FUNCTION_BLOCK FB_MotorCoilsCtrl
VAR_INPUT
	i_Interlocks		:ARRAY[1..8] OF BOOL;
	i_AutoCmdSlow		:BOOL;
	i_AutoCmdFast		:BOOL;
	i_ManCmdSlow		:BOOL;
	i_ManCmdFast		:BOOL;
	i_ManStop			:BOOL;
	i_SlowSpeed			:REAL;
	i_FastSpeed			:REAL;
	i_Feedback1AP		:REAL;
	i_Feedback2AP		:REAL;
	i_EnableMonitor		:BOOL;
	i_MonitorTime		:INT;
	i_MonitorTolerance	:INT;
	i_ServiceMode		:BOOL;
	i_MaintLimit		:REAL;
	i_PresetValue		:REAL;
	i_WritePreset		:BOOL;
END_VAR
VAR_OUTPUT
	q_InterlocksOK		:BOOL;
	q_bCmdSlow			:BOOL;
	q_bCmdFast			:BOOL;
	q_FeedbackMonFlt	:BOOL;
	q_TotalHours		:REAL;
	q_MaintHours		:REAL;
	q_bMaintCall		:BOOL;	
	q_State				:INT;
END_VAR
VAR
	bInTolerance		:BOOL;
	tRunTime			:TIME;
	rRunTime			:REAL;
	tonMonFdb			:TON;
	tonMotorRun			:TON;
	tofMotorRun			:TOF;
END_VAR
VAR // added by the converter: edge detectors and wires of the graphical bodies
    _w1, _w2 : BOOL;
    _ft1, _ft2 : F_TRIG;
    _rt1 : R_TRIG;
END_VAR

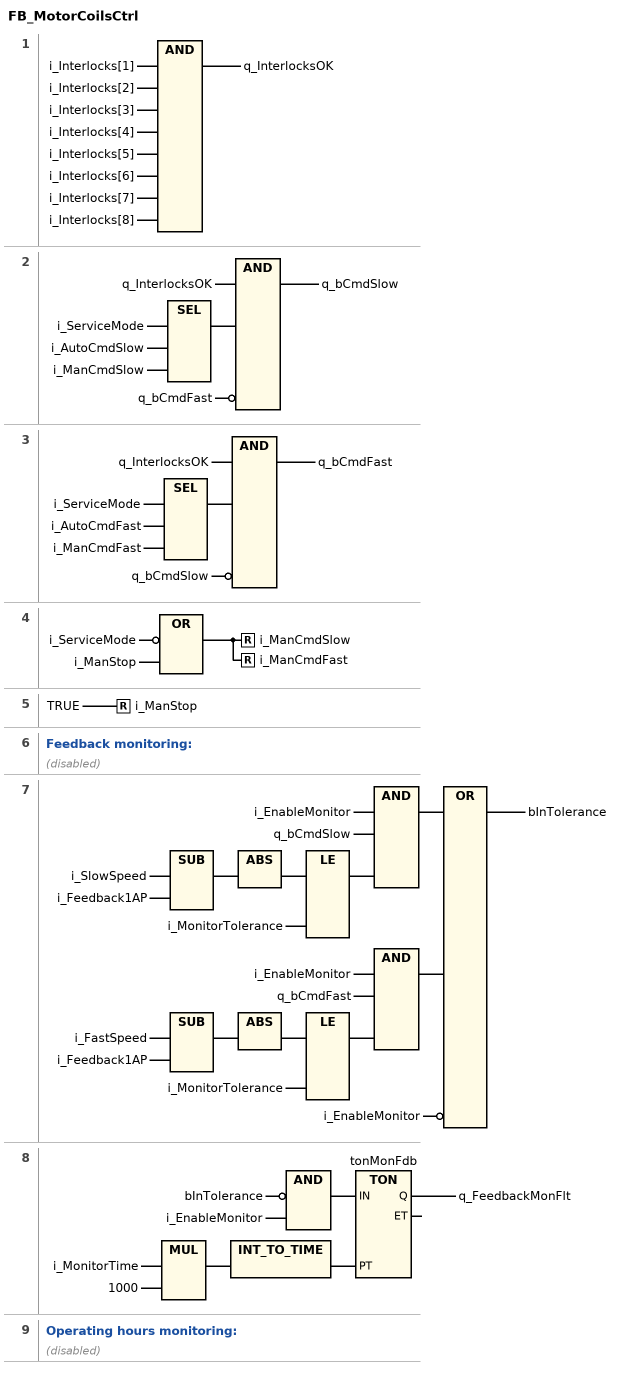
// NETWORK 1
q_InterlocksOK := i_Interlocks[1] AND i_Interlocks[2] AND i_Interlocks[3] AND i_Interlocks[4] AND i_Interlocks[5] AND i_Interlocks[6] AND i_Interlocks[7] AND i_Interlocks[8];

// NETWORK 2
q_bCmdSlow := q_InterlocksOK AND SEL(i_ServiceMode, i_AutoCmdSlow, i_ManCmdSlow) AND NOT q_bCmdFast;

// NETWORK 3
q_bCmdFast := q_InterlocksOK AND SEL(i_ServiceMode, i_AutoCmdFast, i_ManCmdFast) AND NOT q_bCmdSlow;

// NETWORK 4
_w1 := NOT i_ServiceMode OR i_ManStop;
i_ManCmdSlow R= _w1;
i_ManCmdFast R= _w1;

// NETWORK 5
i_ManStop R= TRUE;

// NETWORK 6 (disabled)
// label: Feedback monitoring

// NETWORK 7
bInTolerance := i_EnableMonitor AND q_bCmdSlow AND ABS(i_SlowSpeed - i_Feedback1AP) <= i_MonitorTolerance OR i_EnableMonitor AND q_bCmdFast AND ABS(i_FastSpeed - i_Feedback1AP) <= i_MonitorTolerance OR NOT i_EnableMonitor;

// NETWORK 8
tonMonFdb(IN := NOT bInTolerance AND i_EnableMonitor, PT := INT_TO_TIME(i_MonitorTime * 1000)); // TON
q_FeedbackMonFlt := tonMonFdb.Q;

// NETWORK 9 (disabled)
// label: Operating hours monitoring

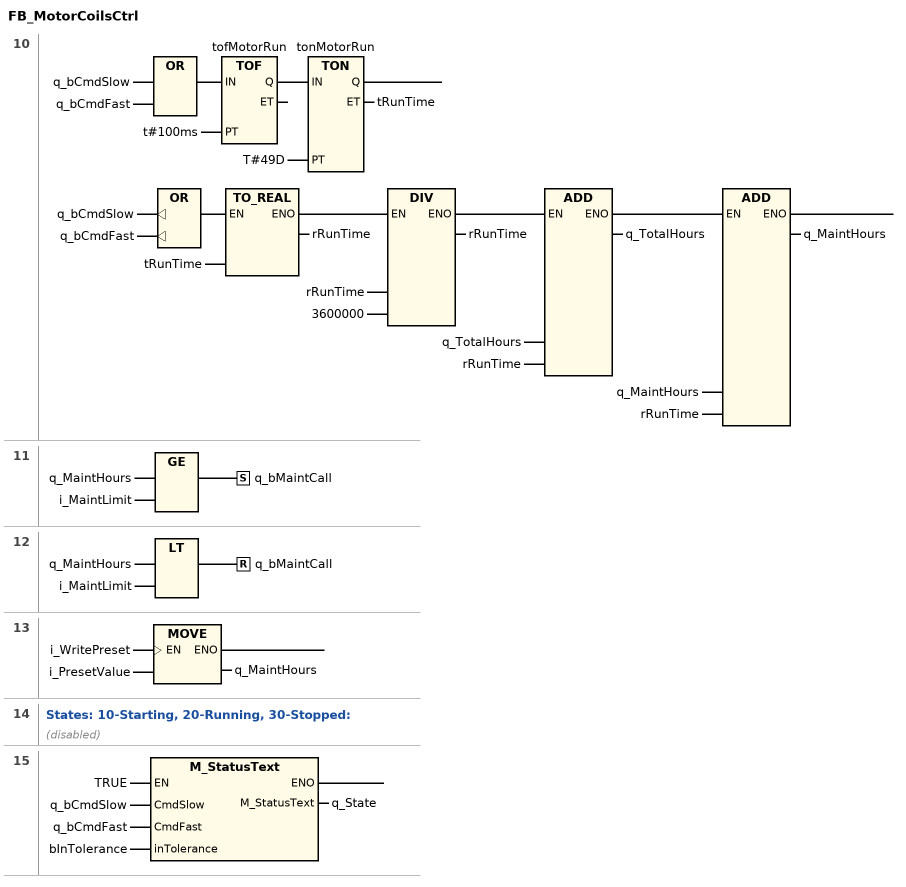
// NETWORK 10
tofMotorRun(IN := q_bCmdSlow OR q_bCmdFast, PT := t#100ms); // TOF
tonMotorRun(IN := tofMotorRun.Q, PT := T#49D, ET => tRunTime); // TON
_ft1(CLK := q_bCmdSlow);
_ft2(CLK := q_bCmdFast);
_w2 := _ft1.Q OR _ft2.Q;
IF _w2 THEN rRunTime := TO_REAL(tRunTime); END_IF
IF _w2 THEN rRunTime := rRunTime / 3600000; END_IF
IF _w2 THEN q_TotalHours := q_TotalHours + rRunTime; END_IF
IF _w2 THEN q_MaintHours := q_MaintHours + rRunTime; END_IF

// NETWORK 11
q_bMaintCall S= q_MaintHours >= i_MaintLimit;

// NETWORK 12
q_bMaintCall R= q_MaintHours < i_MaintLimit;

// NETWORK 13
_rt1(CLK := i_WritePreset);
IF _rt1.Q THEN q_MaintHours := i_PresetValue; END_IF

// NETWORK 14 (disabled)
// label: States: 10-Starting, 20-Running, 30-Stopped

// NETWORK 15
q_State := M_StatusText(CmdSlow := q_bCmdSlow, CmdFast := q_bCmdFast, inTolerance := bInTolerance);

METHOD M_StatusText : INT
VAR_INPUT
	CmdSlow		:BOOL;
	CmdFast		:BOOL;
	inTolerance	:BOOL;
END_VAR
IF (CmdSlow OR CmdFast) AND NOT inTolerance THEN
	M_StatusText := 10;	//Starting
ELSIF (CmdSlow OR CmdFast) AND inTolerance THEN
	M_StatusText := 20;	//Running
ELSIF (NOT CmdSlow AND NOT CmdFast) THEN
	M_StatusText := 30;	//Stopped
END_IF
END_METHOD

END_FUNCTION_BLOCK

(* stored: Version 1.1.0.1, ProductVersion 3.1.4024.12
   POU FB_MotorCoilsCtrl: Id {a90798de-8e56-4b7b-88ed-c025baf0e566}, SpecialFunc None
   Method M_StatusText: Id {b5a103fd-a5af-40f6-9981-2bb98509d6ad} *)
